{attribute addProperty BoxType "BK1250-0000-0000"}
{attribute addProperty Id "CouplerStateAT %I*UINT000"}
{attribute addProperty CRC "1862631496"}
{attribute addProperty SizeInBites "0"}
{attribute addProperty SizeInBytes "0"}
TYPE Inputs_6F058048 :
STRUCT
	{attribute addProperty Name "CouplerState"}
	CouplerState AT %I* : UINT;
END_STRUCT
END_TYPE

(* stored: Version 1.2.0.0, ProductVersion 3.1.4024.9
   DUT Inputs_6F058048: Id {868a5f49-bfec-4c06-a54e-230da71b2b25} *)
